FUNCTION_BLOCK RpcManager IMPLEMENTS I_RpcManager
VAR
	syncRpcHandlers : I_SynchronousRpcHandlers;
	asyncRpcHandlers : I_AsynchronousRpcHandlers;
	asyncResponseManager : I_AsyncResponseManager;
	headerAccessor : I_RpcHeaderAccessor;
	asyncRpcCallQueue : I_AsyncRpcCallQueue;
END_VAR

METHOD FB_init : BOOL
VAR_INPUT
	bInitRetains : BOOL; // if TRUE, the retain variables are initialized (warm start / cold start)
	bInCopyCode : BOOL;  // if TRUE, the instance afterwards gets moved into the copy code (online change)
	SyncRpcHandlers : I_SynchronousRpcHandlers;
	AsyncRpcHandlers : I_AsynchronousRpcHandlers;
	AsyncResponseManager : I_AsyncResponseManager;
	HeaderAccessor : I_RpcHeaderAccessor;
	AsyncRpcCallQueue : I_AsyncRpcCallQueue;
END_VAR
THIS^.syncRpcHandlers := SyncRpcHandlers;
THIS^.asyncRpcHandlers := AsyncRpcHandlers;
THIS^.asyncResponseManager := AsyncResponseManager;
THIS^.headerAccessor := HeaderAccessor;
THIS^.asyncRpcCallQueue := asyncRpcCallQueue;
END_METHOD

METHOD PROTECTED HandleAsyncRpcRequest
VAR_INPUT
	Request : I_Request;
	Response : I_ServerResponse;
	Handler : I_AsynchronousRpcHandler;
END_VAR
VAR
	deserializer : I_Deserializer;
	serializer : I_Serializer;
	asynchronousRpcResponse : I_AsynchronousRpcResponse;
END_VAR
IF NOT TryCreateSerializer(Request, serializer) THEN
	Response.Error('INVALID_HEADER_ACCEPT_TYPE', 'Missing or unsupported accept type in header');
	RETURN;
END_IF

IF NOT TryCreateDeserializer(Request, deserializer) THEN
	Response.Error('INVALID_HEADER_CONTENT_TYPE','Missing or unsupported content type in header');
	serializer.Dispose();
	RETURN;
END_IF

IF NOT TryCreateAsynchronousRpcResponse(Response, serializer, asynchronousRpcResponse) THEN
	Response.Error('SERVER_INTERNAL_ERROR','Unable to create asynchronous response for handler');
	serializer.Dispose();
	deserializer.Dispose();
	RETURN;
END_IF

IF NOT asyncRpcCallQueue.TryAddRpcCall(deserializer, asynchronousRpcResponse, Handler) THEN
	serializer.Dispose();
	deserializer.Dispose();
	asynchronousRpcResponse.RejectWithError('SERVER_INTERNAL_ERROR','Unable to create rpc call');
	RETURN;
END_IF

// we can dispose of the serializer at this stage as it was only used as a prototype.
// this is because when the asynchronousRpcResponse is created then it clones it's serializer. 
serializer.Dispose();
END_METHOD

METHOD PROTECTED HandleSyncRpcRequest
VAR_INPUT
	Request : I_Request;
	Response : I_ServerResponse;
	Handler : I_SynchronousRpcHandler;
END_VAR
VAR
	deserializer : I_Deserializer;
	serializer : I_Serializer;
	synchronousRpcResponse : I_SynchronousRpcResponse;
END_VAR
IF NOT TryCreateSerializer(Request, serializer) THEN
	Response.Error('INVALID_HEADER_ACCEPT_TYPE','Missing or unsupported accept type in header');
	RETURN;
END_IF

IF NOT TryCreateDeserializer(Request, deserializer) THEN
	Response.Error('INVALID_HEADER_CONTENT_TYPE','Missing or unsupported content type in header');
	serializer.Dispose();
	RETURN;
END_IF

IF NOT TryCreateSynchronousRpcResponse(Response, serializer, synchronousRpcResponse) THEN
	Response.Error('SERVER_INTERNAL_ERROR','Unable to create synchronous response for handler');
	serializer.Dispose();
	deserializer.Dispose();
	RETURN;
END_IF

Handler.Handle(deserializer, synchronousRpcResponse);

synchronousRpcResponse.Dispose();
deserializer.Dispose();
serializer.Dispose();

IF NOT Response.HeadersSent THEN
	Response.Error('SERVER_INTERNAL_ERROR','Handler did not return a valid response');
	RETURN;
END_IF
END_METHOD

METHOD PROTECTED TryCreateAsynchronousRpcResponse : BOOL
VAR_INPUT
	Response : I_ServerResponse;
	ResponseSerializer : I_Serializer;
	Destination : REFERENCE TO I_AsynchronousRpcResponse;
END_VAR
VAR
	asynchronousRpcResponseFactory : AsynchronousRpcResponseFactory(Response, ResponseSerializer, asyncResponseManager);
END_VAR
IF Response = 0 THEN 
	RETURN;
END_IF

IF ResponseSerializer = 0 THEN
	RETURN;
END_IF

TryCreateAsynchronousRpcResponse := asynchronousRpcResponseFactory.TryCreate(Destination);
END_METHOD

METHOD PROTECTED TryCreateDeserializer : BOOL
VAR_INPUT
	Request : I_Request;
	Destination : REFERENCE TO I_Deserializer;
END_VAR
VAR
	contentType : T_MAXSTRING;
	pJsonDeserializer : POINTER TO JsonDeserializer;
	pJson : POINTER TO STRING;
END_VAR
IF NOT(headerAccessor.TryGetContentTypeFromRequest(Request, contentType)) THEN
	// unlike TryCreateSerializer, a content type must be included.  Therefore if it 
	// is missing a fault will be raised and the request will be rejected.
	RETURN;
END_IF

IF contentType = headerAccessor.ContentType_Json THEN
	pJsonDeserializer := __NEW(JsonDeserializer);
	pJson := request.PayloadAddress;
	pJsonDeserializer^.TryLoad(pJson^);
	
	Destination := pJsonDeserializer^;
	TryCreateDeserializer := TRUE;
	RETURN;
END_IF

// add other supported formats here...
END_METHOD

METHOD PROTECTED TryCreateSerializer : BOOL
VAR_INPUT
	Request : I_Request;
	Destination : REFERENCE TO I_Serializer;
END_VAR
VAR
	acceptType : T_MAXSTRING;
	pJsonSerializer : POINTER TO JsonSerializer;
END_VAR
IF NOT(headerAccessor.TryGetAcceptResponseFormatFromRequest(Request, acceptType)) THEN
	// if no header is provided for the accept type, then the line below selects the default return type. 
	// change this line to change the default.
	acceptType := headerAccessor.ContentType_Json;
END_IF

IF acceptType = headerAccessor.ContentType_Json THEN
	pJsonSerializer := __NEW(JsonSerializer);
	Destination := pJsonSerializer^;
	TryCreateSerializer := TRUE;
	RETURN;
END_IF

// add other supported formats here...
END_METHOD

METHOD PROTECTED TryCreateSynchronousRpcResponse : BOOL
VAR_INPUT
	Response : I_ServerResponse;
	ResponseSerializer : I_Serializer;
	Destination : REFERENCE TO I_SynchronousRpcResponse;
END_VAR
VAR
	pSynchronousRpcResponse : POINTER TO SynchronousRpcResponse;
END_VAR
IF Response = 0 THEN 
	RETURN;
END_IF

IF ResponseSerializer = 0 THEN
	RETURN;
END_IF

pSynchronousRpcResponse := __NEW(SynchronousRpcResponse(ServerResponse := Response, Serializer := ResponseSerializer, AsyncResponseManager := THIS^.asyncResponseManager));
Destination := pSynchronousRpcResponse^;
TryCreateSynchronousRpcResponse := TRUE;
END_METHOD

METHOD PUBLIC TryHandleIncomingRequest : BOOL
VAR_INPUT
	Request : I_Request;
	Response : I_ServerResponse;
END_VAR
VAR
	requestType : T_MAXSTRING;
	methodName : T_MAXSTRING;
	asyncRpcHandler : I_AsynchronousRpcHandler;
	syncRpcHandler : I_SynchronousRpcHandler;
END_VAR
IF NOT headerAccessor.TryGetTypeFromRequest(Request, requestType) THEN
	RETURN;
END_IF

IF requestType <> 'RPC 1.0' THEN
	RETURN;
END_IF

IF NOT headerAccessor.TryGetMethodNameFromRequest(Request, methodName) THEN
	Response.Error('INVALID_RPC_METHOD_NAME','Missing RPC method name');
	TryHandleIncomingRequest := TRUE;
	RETURN;
END_IF

IF asyncRpcHandlers.hasHandlers AND_THEN asyncRpcHandlers.TryGetByMethodName(methodName, asyncRpcHandler) THEN
	HandleAsyncRpcRequest(Request, Response, asyncRpcHandler);
	TryHandleIncomingRequest := TRUE;
	RETURN;
END_IF

IF syncRpcHandlers.hasHandlers AND_THEN syncRpcHandlers.TryGetByMethodName(methodName, syncRpcHandler) THEN
	HandleSyncRpcRequest(Request, Response, syncRpcHandler);
	TryHandleIncomingRequest := TRUE;
	RETURN;
END_IF
END_METHOD

END_FUNCTION_BLOCK

(* stored: Version 1.1.0.1, ProductVersion 3.1.4024.15
   POU RpcManager: Id {308b5439-3f52-0c22-3a38-2a4336aefe7b}, SpecialFunc None
   Folder Constructor: Id {0ade8a4f-3476-019d-0aba-82e2bb43a90e}
   Folder Protected: Id {fab3162a-e063-4acd-95f5-ec6e3d87a5b3}
   Method FB_init: Id {02d294c0-1ef3-0764-007b-c1c7ca225b00}
   Method HandleAsyncRpcRequest: Id {562f6f63-856d-4ff4-b0d7-f252939359d1}
   Method HandleSyncRpcRequest: Id {c4943403-c364-48b4-88ea-745865db1799}
   Method TryCreateAsynchronousRpcResponse: Id {1b643550-ad2d-40c5-9a58-e6764736bfa0}
   Method TryCreateDeserializer: Id {dedcba2e-7a09-4036-89b7-5f55359564d4}
   Method TryCreateSerializer: Id {afb070c4-4677-4a46-8796-2375baadff3a}
   Method TryCreateSynchronousRpcResponse: Id {c96fe62f-2f56-4271-b9bf-4d2d13323aff}
   Method TryHandleIncomingRequest: Id {b9b37eb6-3223-0f27-2d3b-8d09875b1965} *)
